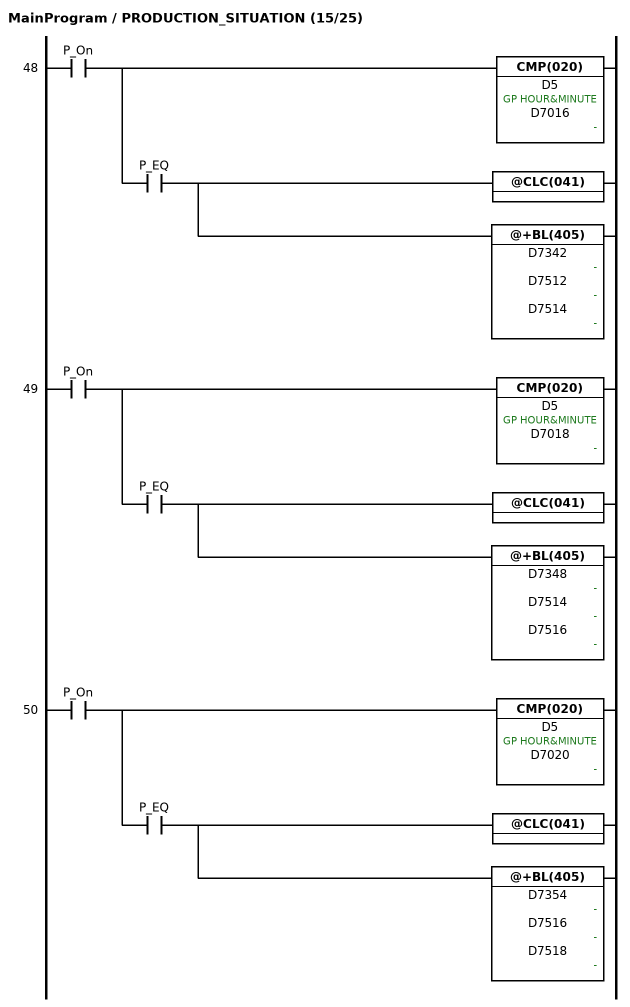
; [picture p240: MainProgram / PRODUCTION_SITUATION, rungs 48-50]
; rung 48
LD P_On
CMP(020) D5 D7016  ; GP HOUR&MINUTE, -
AND P_EQ
@CLC(041)
@+BL(405) D7342 D7512 D7514  ; -
; rung 49
LD P_On
CMP(020) D5 D7018  ; GP HOUR&MINUTE, -
AND P_EQ
@CLC(041)
@+BL(405) D7348 D7514 D7516  ; -
; rung 50
LD P_On
CMP(020) D5 D7020  ; GP HOUR&MINUTE, -
AND P_EQ
@CLC(041)
@+BL(405) D7354 D7516 D7518  ; -

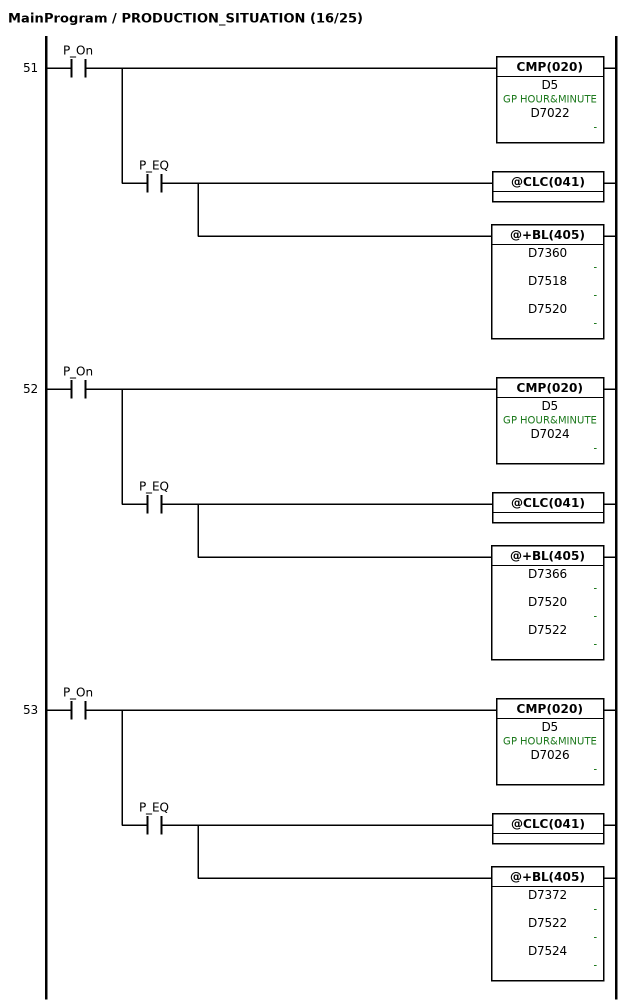
; rung 51
LD P_On
CMP(020) D5 D7022  ; GP HOUR&MINUTE, -
AND P_EQ
@CLC(041)
@+BL(405) D7360 D7518 D7520  ; -
; rung 52
LD P_On
CMP(020) D5 D7024  ; GP HOUR&MINUTE, -
AND P_EQ
@CLC(041)
@+BL(405) D7366 D7520 D7522  ; -
; rung 53
LD P_On
CMP(020) D5 D7026  ; GP HOUR&MINUTE, -
AND P_EQ
@CLC(041)
@+BL(405) D7372 D7522 D7524  ; -

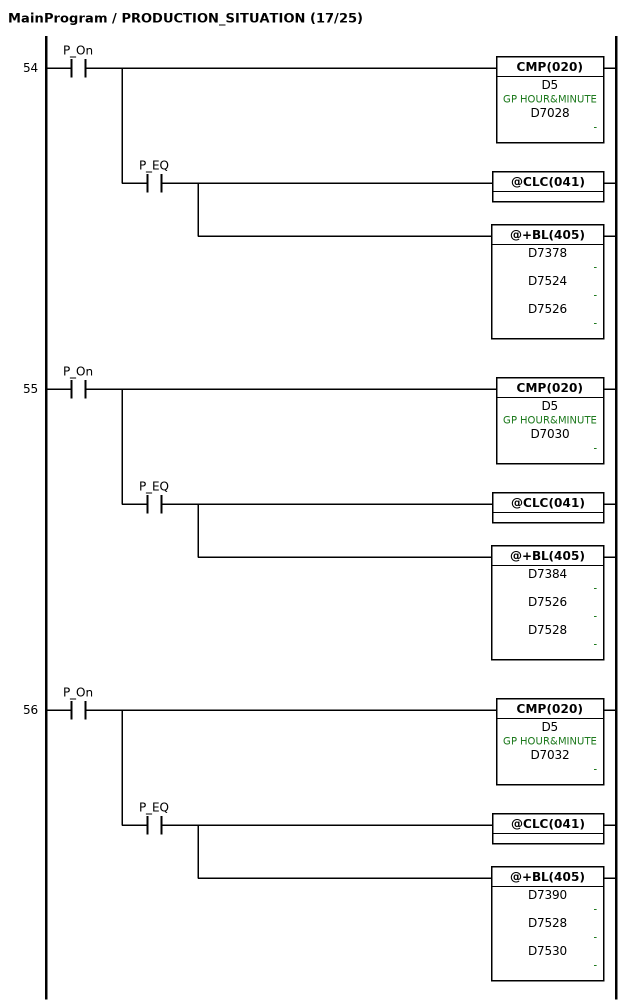
; rung 54
LD P_On
CMP(020) D5 D7028  ; GP HOUR&MINUTE, -
AND P_EQ
@CLC(041)
@+BL(405) D7378 D7524 D7526  ; -
; rung 55
LD P_On
CMP(020) D5 D7030  ; GP HOUR&MINUTE, -
AND P_EQ
@CLC(041)
@+BL(405) D7384 D7526 D7528  ; -
; rung 56
LD P_On
CMP(020) D5 D7032  ; GP HOUR&MINUTE, -
AND P_EQ
@CLC(041)
@+BL(405) D7390 D7528 D7530  ; -

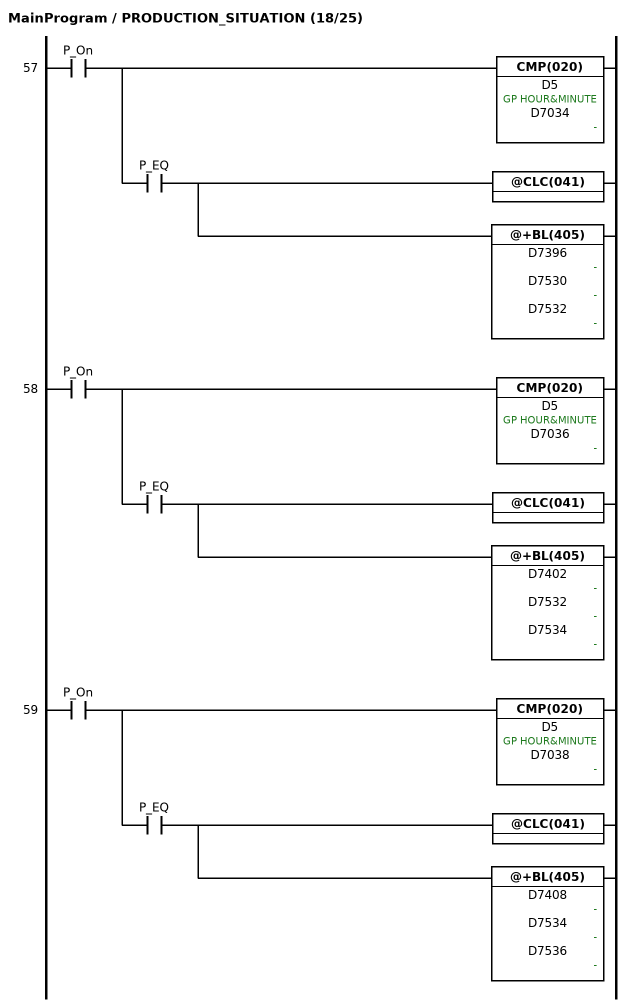
; rung 57
LD P_On
CMP(020) D5 D7034  ; GP HOUR&MINUTE, -
AND P_EQ
@CLC(041)
@+BL(405) D7396 D7530 D7532  ; -
; rung 58
LD P_On
CMP(020) D5 D7036  ; GP HOUR&MINUTE, -
AND P_EQ
@CLC(041)
@+BL(405) D7402 D7532 D7534  ; -
; rung 59
LD P_On
CMP(020) D5 D7038  ; GP HOUR&MINUTE, -
AND P_EQ
@CLC(041)
@+BL(405) D7408 D7534 D7536  ; -

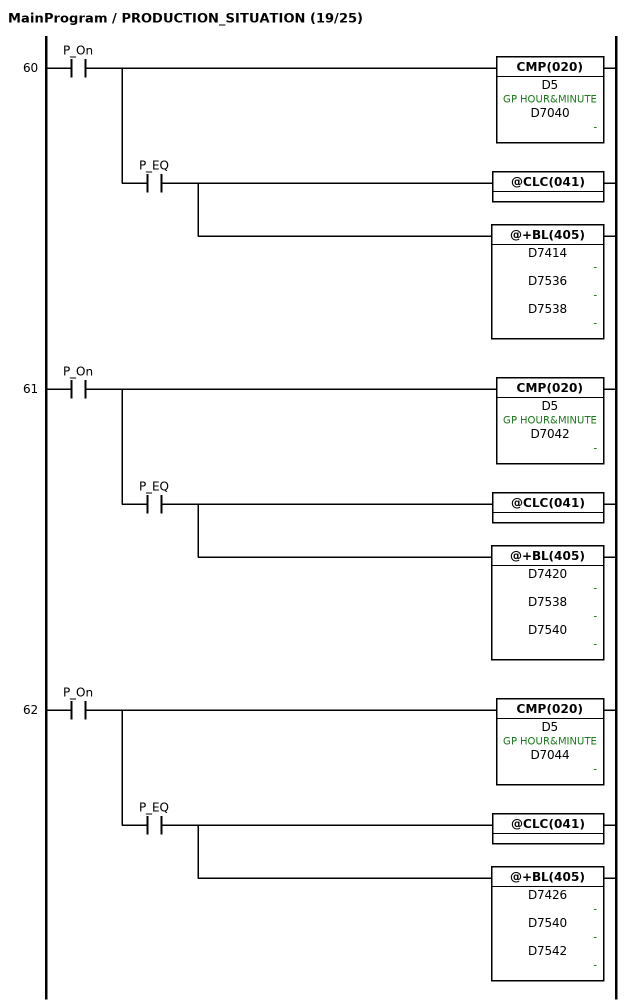
; rung 60
LD P_On
CMP(020) D5 D7040  ; GP HOUR&MINUTE, -
AND P_EQ
@CLC(041)
@+BL(405) D7414 D7536 D7538  ; -
; rung 61
LD P_On
CMP(020) D5 D7042  ; GP HOUR&MINUTE, -
AND P_EQ
@CLC(041)
@+BL(405) D7420 D7538 D7540  ; -
; rung 62
LD P_On
CMP(020) D5 D7044  ; GP HOUR&MINUTE, -
AND P_EQ
@CLC(041)
@+BL(405) D7426 D7540 D7542  ; -

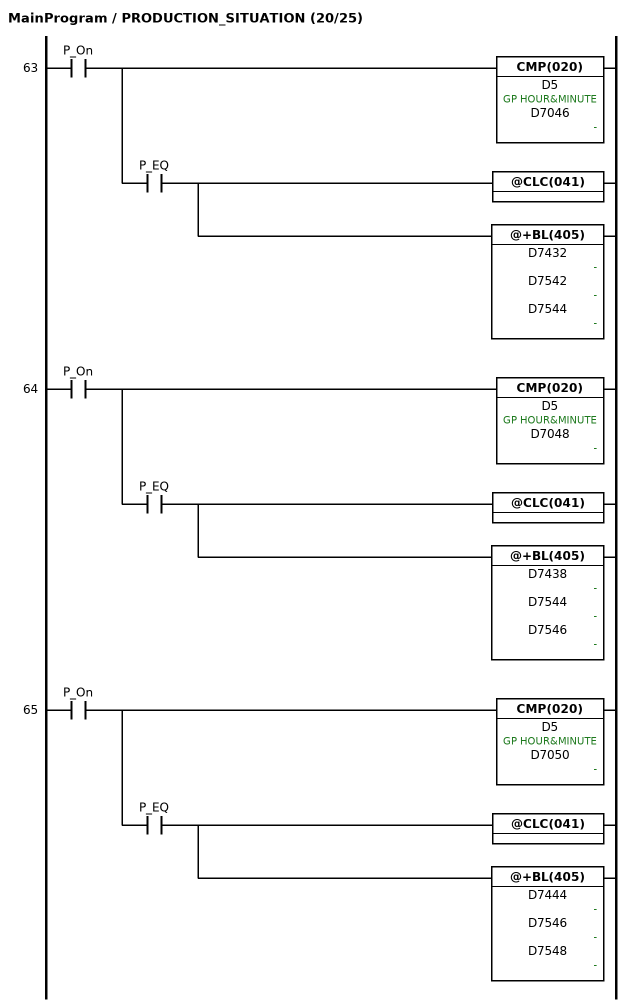
; rung 63
LD P_On
CMP(020) D5 D7046  ; GP HOUR&MINUTE, -
AND P_EQ
@CLC(041)
@+BL(405) D7432 D7542 D7544  ; -
; rung 64
LD P_On
CMP(020) D5 D7048  ; GP HOUR&MINUTE, -
AND P_EQ
@CLC(041)
@+BL(405) D7438 D7544 D7546  ; -
; rung 65
LD P_On
CMP(020) D5 D7050  ; GP HOUR&MINUTE, -
AND P_EQ
@CLC(041)
@+BL(405) D7444 D7546 D7548  ; -

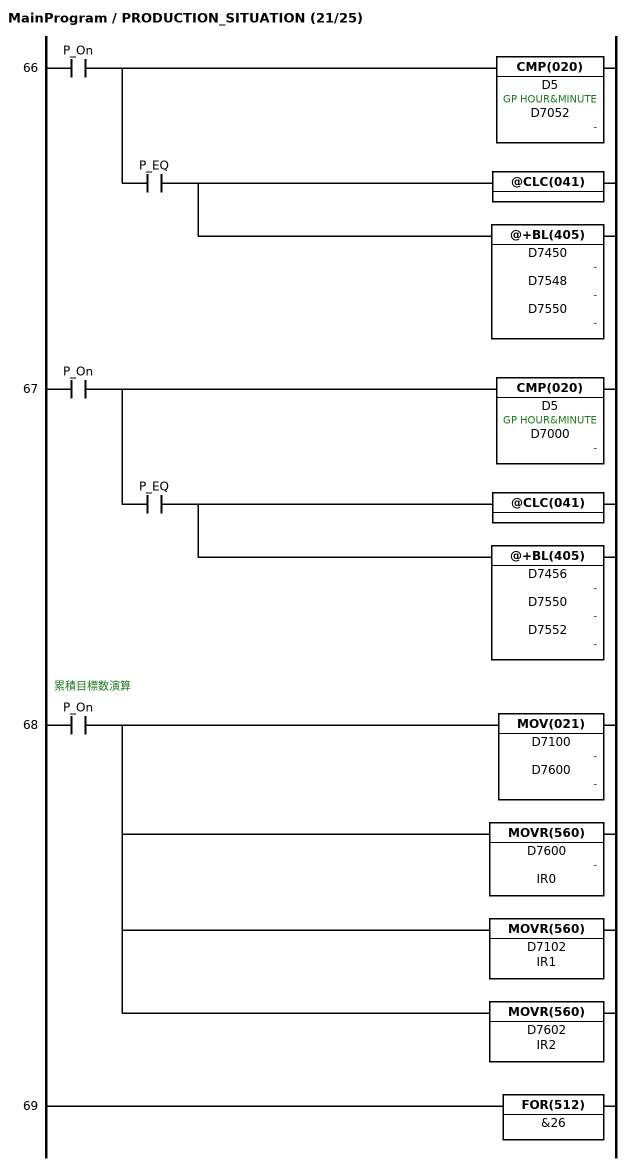
; rung 66
LD P_On
CMP(020) D5 D7052  ; GP HOUR&MINUTE, -
AND P_EQ
@CLC(041)
@+BL(405) D7450 D7548 D7550  ; -
; rung 67
LD P_On
CMP(020) D5 D7000  ; GP HOUR&MINUTE, -
AND P_EQ
@CLC(041)
@+BL(405) D7456 D7550 D7552  ; -
; rung 68: 累積目標数演算
LD P_On
MOV(021) D7100 D7600  ; -
MOVR(560) D7600 IR0  ; -
MOVR(560) D7102 IR1
MOVR(560) D7602 IR2
; rung 69
FOR(512) &26

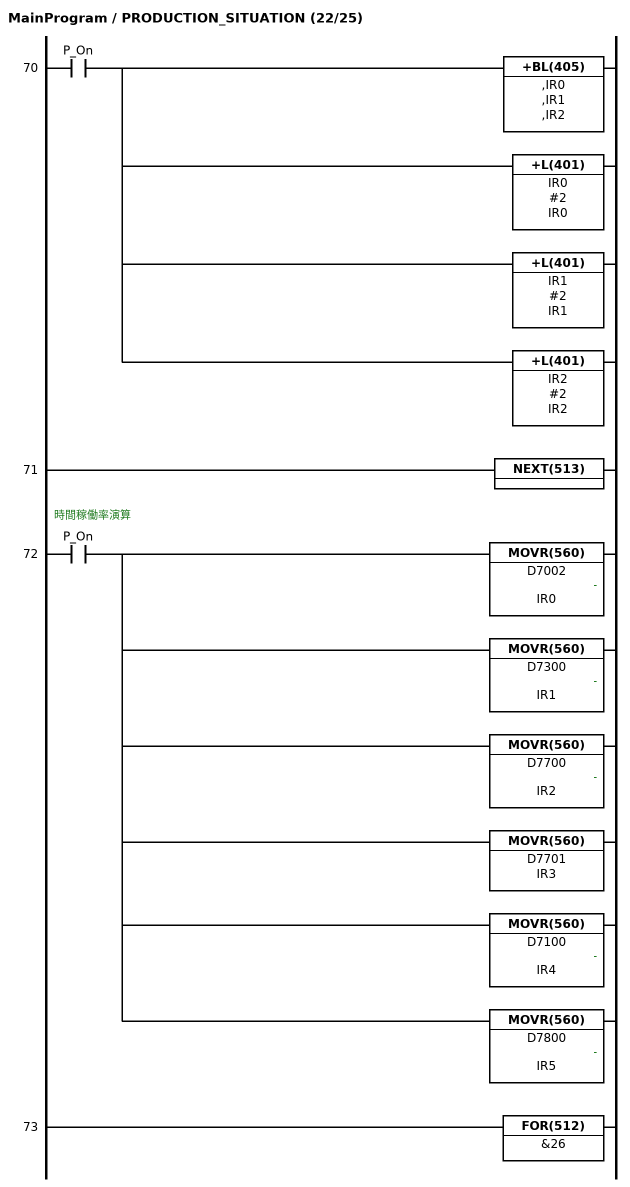
; rung 70
LD P_On
+BL(405) ,IR0 ,IR1 ,IR2
+L(401) IR0 #2 IR0
+L(401) IR1 #2 IR1
+L(401) IR2 #2 IR2
; rung 71
NEXT(513)
; rung 72: 時間稼働率演算
LD P_On
MOVR(560) D7002 IR0  ; -
MOVR(560) D7300 IR1  ; -
MOVR(560) D7700 IR2  ; -
MOVR(560) D7701 IR3
MOVR(560) D7100 IR4  ; -
MOVR(560) D7800 IR5  ; -
; rung 73
FOR(512) &26

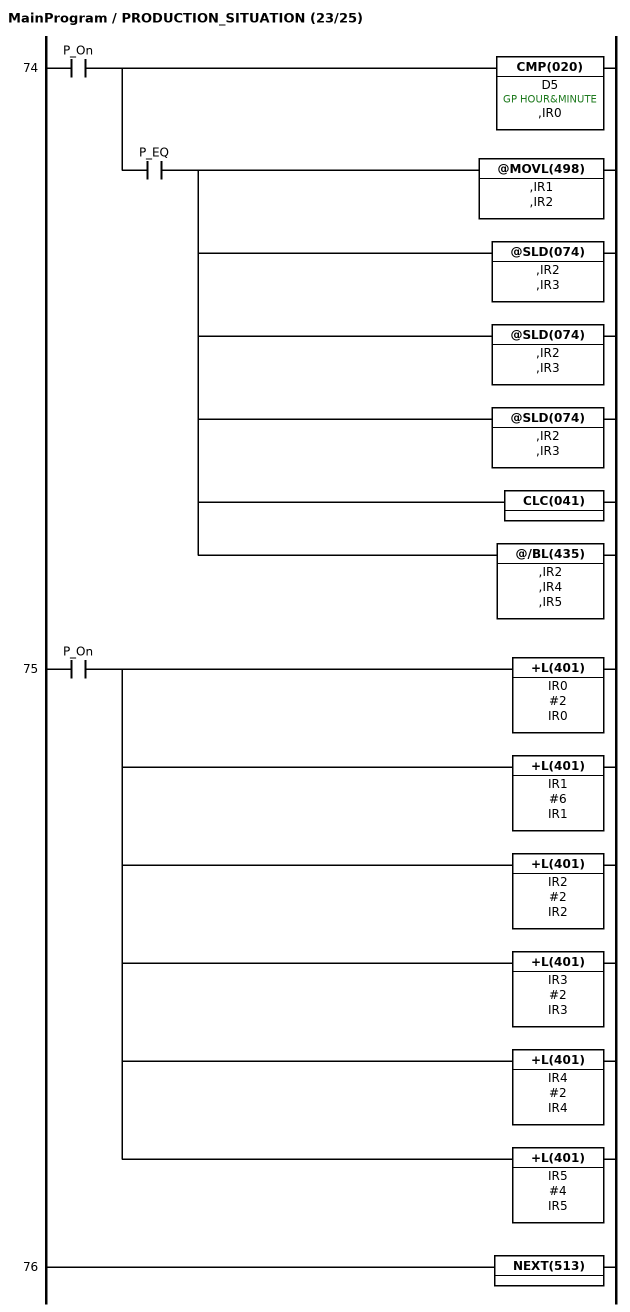
; rung 74
LD P_On
CMP(020) D5 ,IR0  ; GP HOUR&MINUTE
AND P_EQ
@MOVL(498) ,IR1 ,IR2
@SLD(074) ,IR2 ,IR3
@SLD(074) ,IR2 ,IR3
@SLD(074) ,IR2 ,IR3
CLC(041)
@/BL(435) ,IR2 ,IR4 ,IR5
; rung 75
LD P_On
+L(401) IR0 #2 IR0
+L(401) IR1 #6 IR1
+L(401) IR2 #2 IR2
+L(401) IR3 #2 IR3
+L(401) IR4 #2 IR4
+L(401) IR5 #4 IR5
; rung 76
NEXT(513)

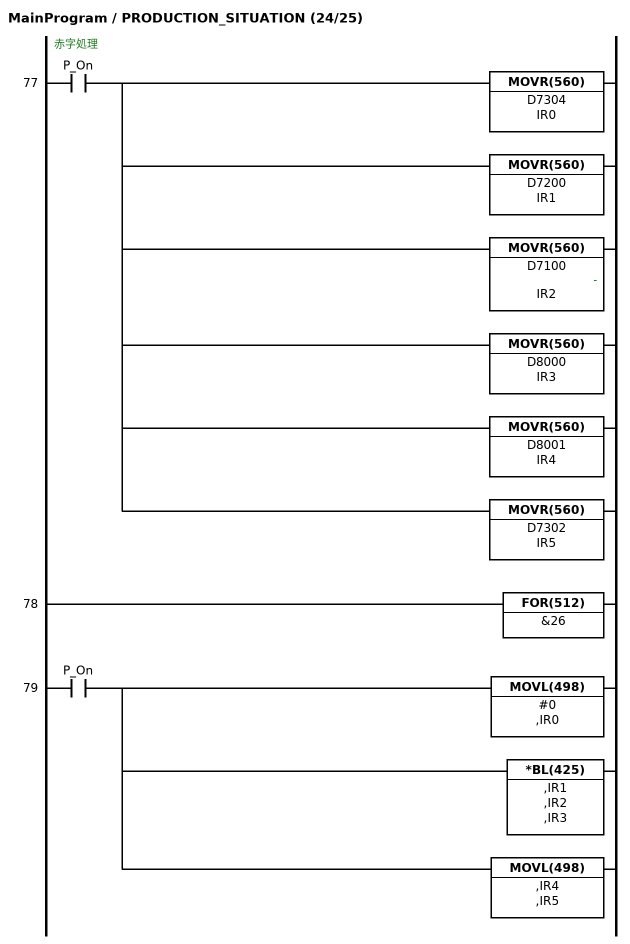
; rung 77: 赤字処理
LD P_On
MOVR(560) D7304 IR0
MOVR(560) D7200 IR1
MOVR(560) D7100 IR2  ; -
MOVR(560) D8000 IR3
MOVR(560) D8001 IR4
MOVR(560) D7302 IR5
; rung 78
FOR(512) &26
; rung 79
LD P_On
MOVL(498) #0 ,IR0
*BL(425) ,IR1 ,IR2 ,IR3
MOVL(498) ,IR4 ,IR5

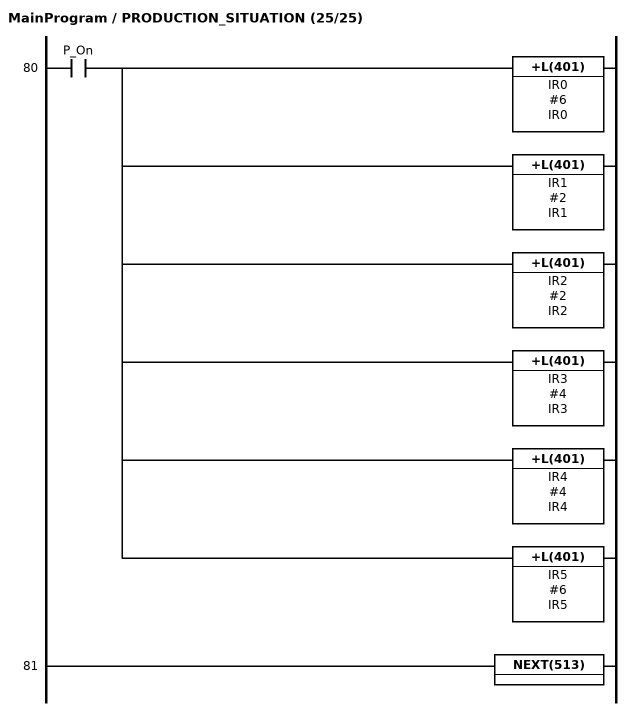
; rung 80
LD P_On
+L(401) IR0 #6 IR0
+L(401) IR1 #2 IR1
+L(401) IR2 #2 IR2
+L(401) IR3 #4 IR3
+L(401) IR4 #4 IR4
+L(401) IR5 #6 IR5
; rung 81
NEXT(513)

### Section OPERATION_RATE

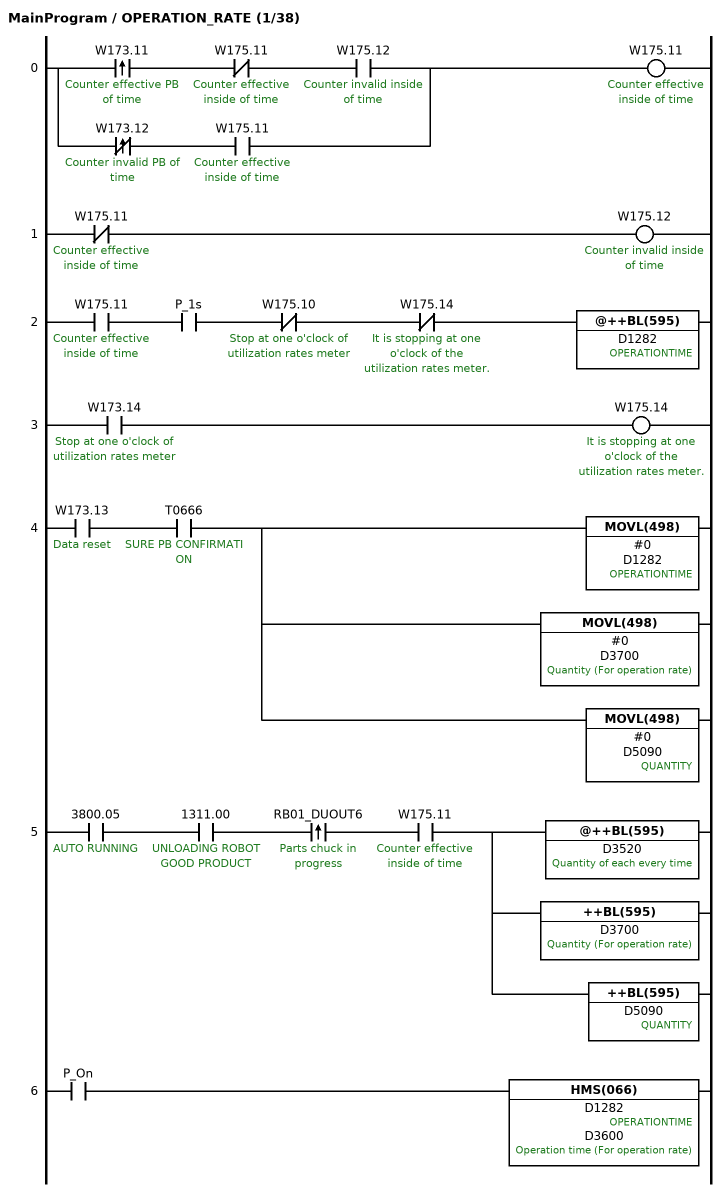
; rung 0
@LD W173.11  ; Counter effective PB of time
ANDNOT W175.11  ; Counter effective inside of time
AND W175.12  ; Counter invalid inside of time
@LDNOT W173.12  ; Counter invalid PB of time
AND W175.11  ; Counter effective inside of time
ORLD
OUT W175.11  ; Counter effective inside of time
; rung 1
LDNOT W175.11  ; Counter effective inside of time
OUT W175.12  ; Counter invalid inside of time
; rung 2
LD W175.11  ; Counter effective inside of time
AND P_1s
ANDNOT W175.10  ; Stop at one o'clock of utilization rates meter
ANDNOT W175.14  ; It is stopping at one o'clock of the utilization rates meter.
@++BL(595) D1282  ; OPERATIONTIME
; rung 3
LD W173.14  ; Stop at one o'clock of utilization rates meter
OUT W175.14  ; It is stopping at one o'clock of the utilization rates meter.
; rung 4
LD W173.13  ; Data reset
AND T0666  ; SURE PB CONFIRMATION
MOVL(498) #0 D1282  ; OPERATIONTIME
MOVL(498) #0 D3700  ; Quantity (For operation rate)
MOVL(498) #0 D5090  ; QUANTITY
; rung 5
LD 3800.05  ; AUTO RUNNING
AND 1311.00  ; UNLOADING ROBOT GOOD PRODUCT
@AND RB01_DUOUT6  ; Parts chuck in progress
AND W175.11  ; Counter effective inside of time
@++BL(595) D3520  ; Quantity of each every time
++BL(595) D3700  ; Quantity (For operation rate)
++BL(595) D5090  ; QUANTITY
; rung 6
LD P_On
HMS(066) D1282 D3600  ; OPERATIONTIME, Operation time (For operation rate)

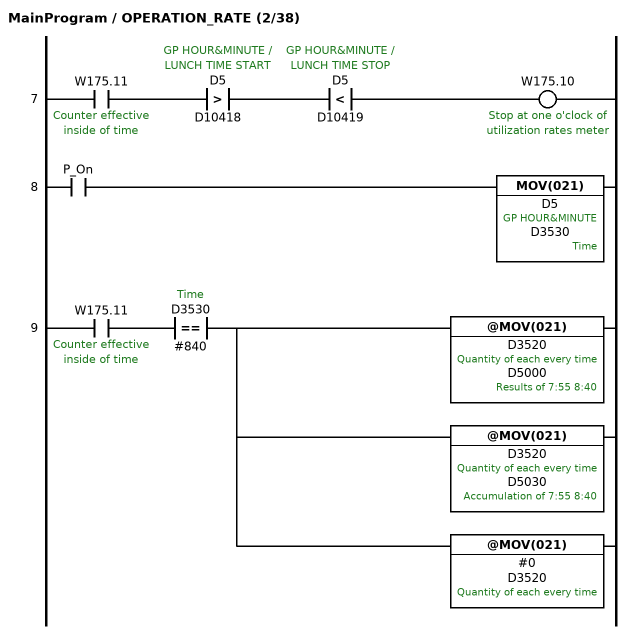
; rung 7
LD W175.11  ; Counter effective inside of time
AND>(320) D5 D10418  ; GP HOUR&MINUTE, LUNCH TIME START
AND<(310) D5 D10419  ; GP HOUR&MINUTE, LUNCH TIME STOP
OUT W175.10  ; Stop at one o'clock of utilization rates meter
; rung 8
LD P_On
MOV(021) D5 D3530  ; GP HOUR&MINUTE, Time
; rung 9
LD W175.11  ; Counter effective inside of time
AND=L(301) D3530 #840  ; Time
@MOV(021) D3520 D5000  ; Quantity of each every time, Results of 7:55 8:40
@MOV(021) D3520 D5030  ; Quantity of each every time, Accumulation of 7:55 8:40
@MOV(021) #0 D3520  ; Quantity of each every time

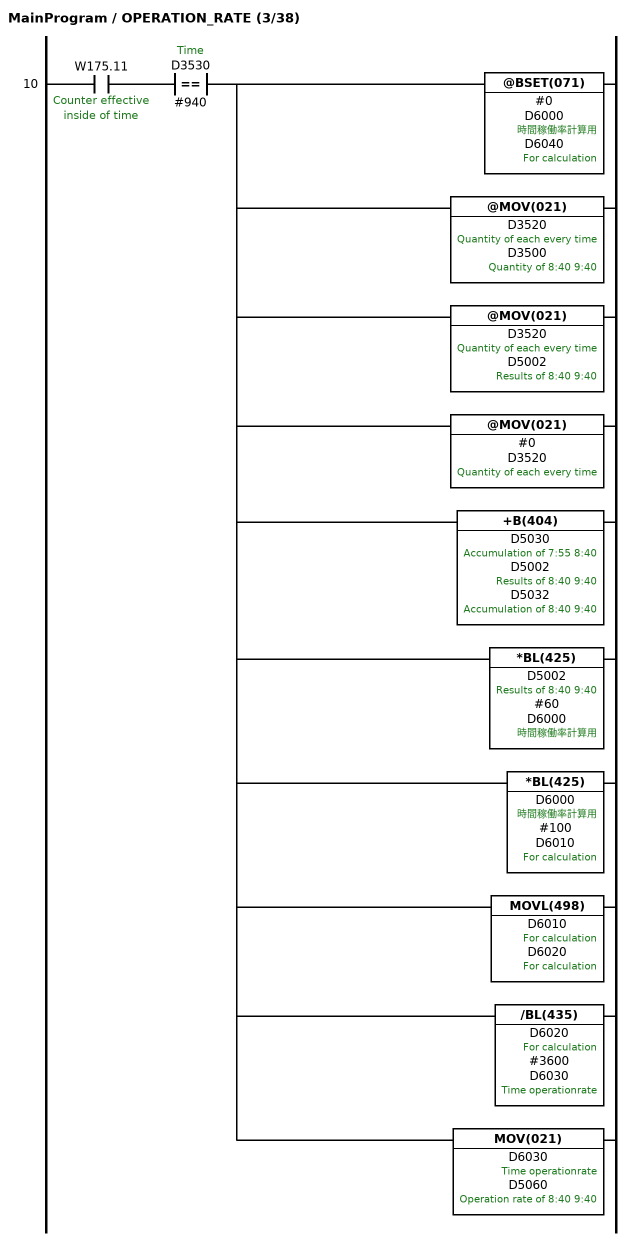
; rung 10
LD W175.11  ; Counter effective inside of time
AND=L(301) D3530 #940  ; Time
@BSET(071) #0 D6000 D6040  ; 時間稼働率計算用, For calculation
@MOV(021) D3520 D3500  ; Quantity of each every time, Quantity of 8:40 9:40
@MOV(021) D3520 D5002  ; Quantity of each every time, Results of 8:40 9:40
@MOV(021) #0 D3520  ; Quantity of each every time
+B(404) D5030 D5002 D5032  ; Accumulation of 7:55 8:40, Results of 8:40 9:40, Accumulation of 8:40 9:40
*BL(425) D5002 #60 D6000  ; Results of 8:40 9:40, 時間稼働率計算用
*BL(425) D6000 #100 D6010  ; 時間稼働率計算用, For calculation
MOVL(498) D6010 D6020  ; For calculation
/BL(435) D6020 #3600 D6030  ; For calculation, Time operationrate
MOV(021) D6030 D5060  ; Time operationrate, Operation rate of 8:40 9:40

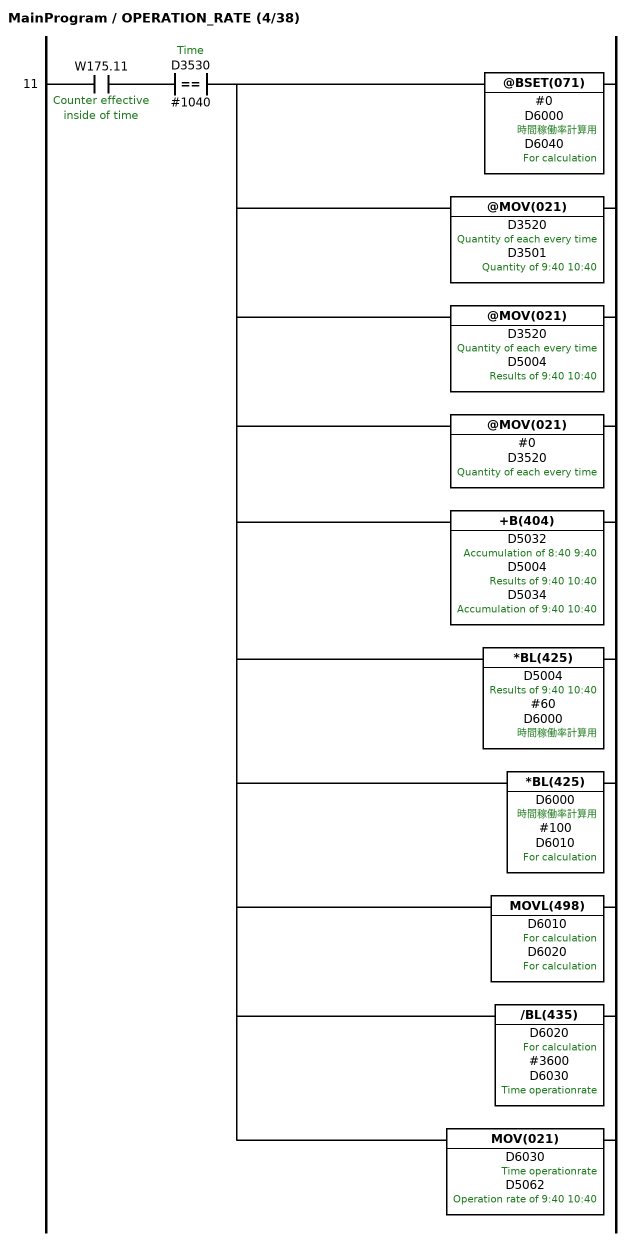
; rung 11
LD W175.11  ; Counter effective inside of time
AND=L(301) D3530 #1040  ; Time
@BSET(071) #0 D6000 D6040  ; 時間稼働率計算用, For calculation
@MOV(021) D3520 D3501  ; Quantity of each every time, Quantity of 9:40 10:40
@MOV(021) D3520 D5004  ; Quantity of each every time, Results of 9:40 10:40
@MOV(021) #0 D3520  ; Quantity of each every time
+B(404) D5032 D5004 D5034  ; Accumulation of 8:40 9:40, Results of 9:40 10:40, Accumulation of 9:40 10:40
*BL(425) D5004 #60 D6000  ; Results of 9:40 10:40, 時間稼働率計算用
*BL(425) D6000 #100 D6010  ; 時間稼働率計算用, For calculation
MOVL(498) D6010 D6020  ; For calculation
/BL(435) D6020 #3600 D6030  ; For calculation, Time operationrate
MOV(021) D6030 D5062  ; Time operationrate, Operation rate of 9:40 10:40

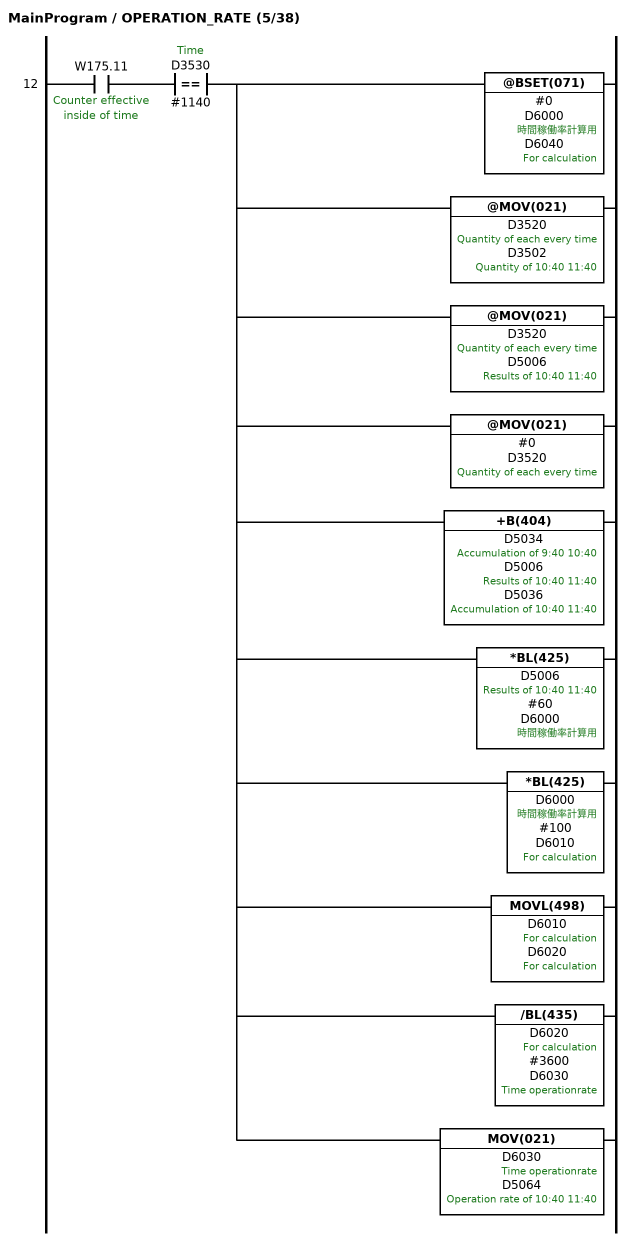
; rung 12
LD W175.11  ; Counter effective inside of time
AND=L(301) D3530 #1140  ; Time
@BSET(071) #0 D6000 D6040  ; 時間稼働率計算用, For calculation
@MOV(021) D3520 D3502  ; Quantity of each every time, Quantity of 10:40 11:40
@MOV(021) D3520 D5006  ; Quantity of each every time, Results of 10:40 11:40
@MOV(021) #0 D3520  ; Quantity of each every time
+B(404) D5034 D5006 D5036  ; Accumulation of 9:40 10:40, Results of 10:40 11:40, Accumulation of 10:40 11:40
*BL(425) D5006 #60 D6000  ; Results of 10:40 11:40, 時間稼働率計算用
*BL(425) D6000 #100 D6010  ; 時間稼働率計算用, For calculation
MOVL(498) D6010 D6020  ; For calculation
/BL(435) D6020 #3600 D6030  ; For calculation, Time operationrate
MOV(021) D6030 D5064  ; Time operationrate, Operation rate of 10:40 11:40

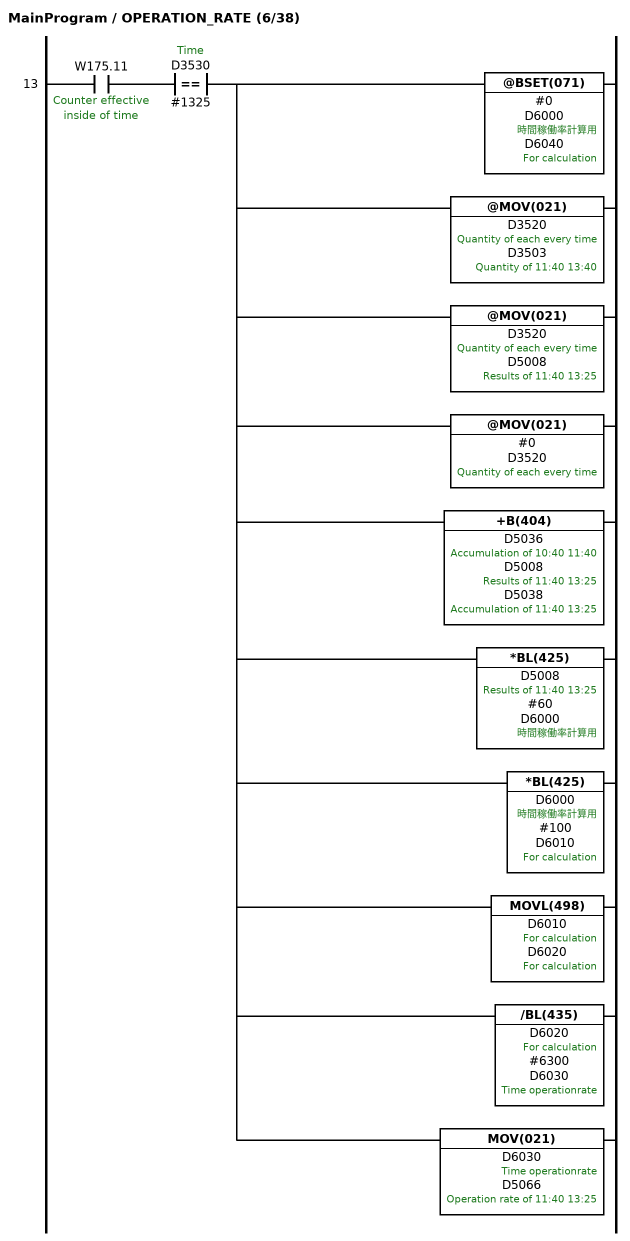
; rung 13
LD W175.11  ; Counter effective inside of time
AND=L(301) D3530 #1325  ; Time
@BSET(071) #0 D6000 D6040  ; 時間稼働率計算用, For calculation
@MOV(021) D3520 D3503  ; Quantity of each every time, Quantity of 11:40 13:40
@MOV(021) D3520 D5008  ; Quantity of each every time, Results of 11:40 13:25
@MOV(021) #0 D3520  ; Quantity of each every time
+B(404) D5036 D5008 D5038  ; Accumulation of 10:40 11:40, Results of 11:40 13:25, Accumulation of 11:40 13:25
*BL(425) D5008 #60 D6000  ; Results of 11:40 13:25, 時間稼働率計算用
*BL(425) D6000 #100 D6010  ; 時間稼働率計算用, For calculation
MOVL(498) D6010 D6020  ; For calculation
/BL(435) D6020 #6300 D6030  ; For calculation, Time operationrate
MOV(021) D6030 D5066  ; Time operationrate, Operation rate of 11:40 13:25

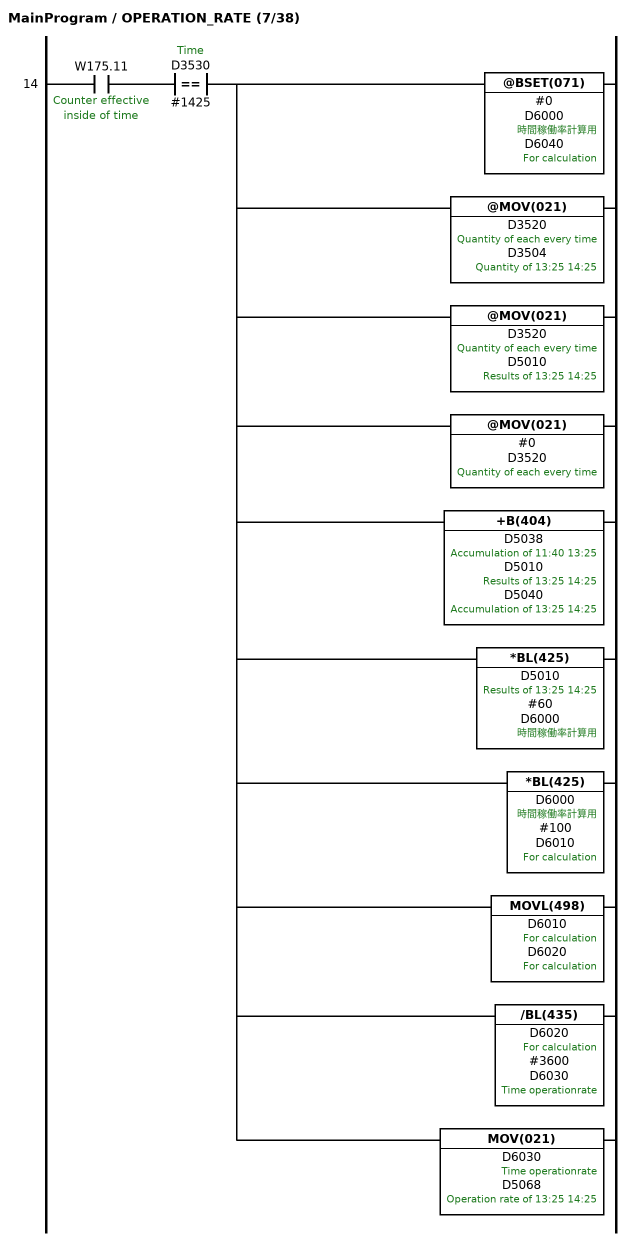
; rung 14
LD W175.11  ; Counter effective inside of time
AND=L(301) D3530 #1425  ; Time
@BSET(071) #0 D6000 D6040  ; 時間稼働率計算用, For calculation
@MOV(021) D3520 D3504  ; Quantity of each every time, Quantity of 13:25 14:25
@MOV(021) D3520 D5010  ; Quantity of each every time, Results of 13:25 14:25
@MOV(021) #0 D3520  ; Quantity of each every time
+B(404) D5038 D5010 D5040  ; Accumulation of 11:40 13:25, Results of 13:25 14:25, Accumulation of 13:25 14:25
*BL(425) D5010 #60 D6000  ; Results of 13:25 14:25, 時間稼働率計算用
*BL(425) D6000 #100 D6010  ; 時間稼働率計算用, For calculation
MOVL(498) D6010 D6020  ; For calculation
/BL(435) D6020 #3600 D6030  ; For calculation, Time operationrate
MOV(021) D6030 D5068  ; Time operationrate, Operation rate of 13:25 14:25

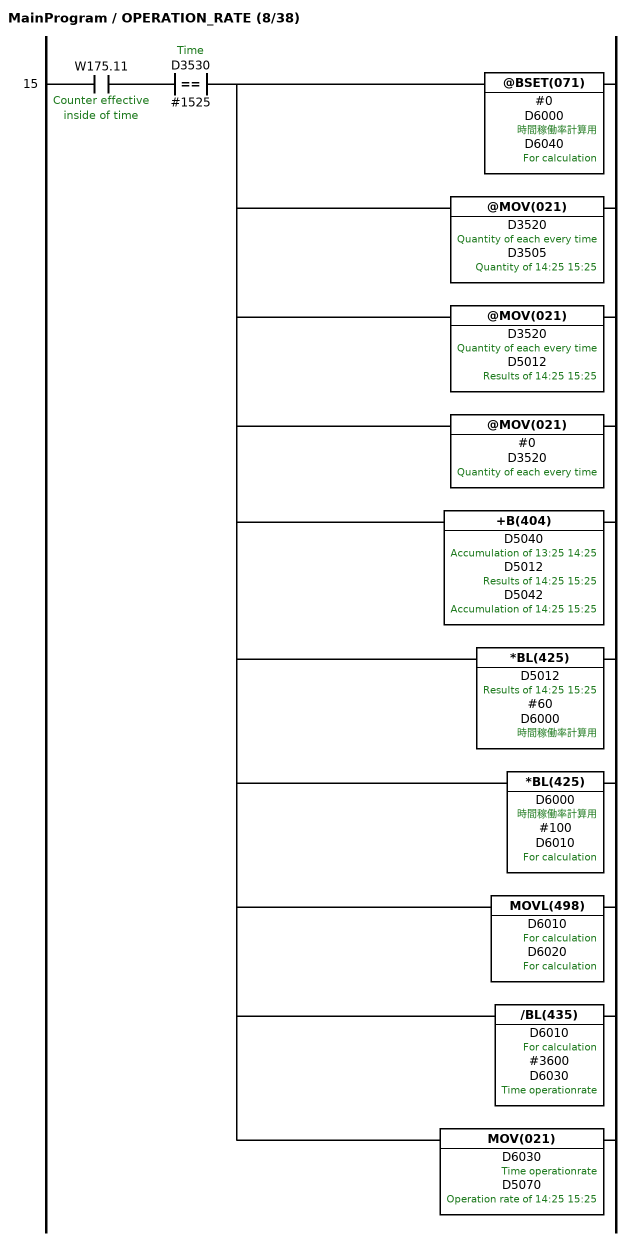
; rung 15
LD W175.11  ; Counter effective inside of time
AND=L(301) D3530 #1525  ; Time
@BSET(071) #0 D6000 D6040  ; 時間稼働率計算用, For calculation
@MOV(021) D3520 D3505  ; Quantity of each every time, Quantity of 14:25 15:25
@MOV(021) D3520 D5012  ; Quantity of each every time, Results of 14:25 15:25
@MOV(021) #0 D3520  ; Quantity of each every time
+B(404) D5040 D5012 D5042  ; Accumulation of 13:25 14:25, Results of 14:25 15:25, Accumulation of 14:25 15:25
*BL(425) D5012 #60 D6000  ; Results of 14:25 15:25, 時間稼働率計算用
*BL(425) D6000 #100 D6010  ; 時間稼働率計算用, For calculation
MOVL(498) D6010 D6020  ; For calculation
/BL(435) D6010 #3600 D6030  ; For calculation, Time operationrate
MOV(021) D6030 D5070  ; Time operationrate, Operation rate of 14:25 15:25

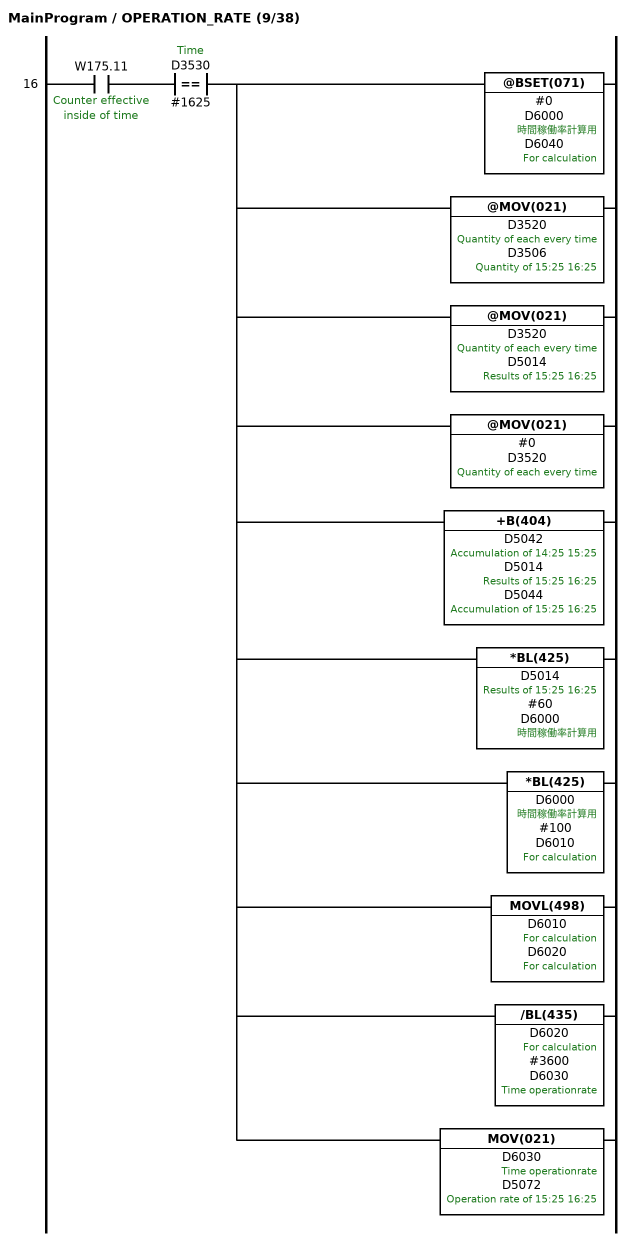
; rung 16
LD W175.11  ; Counter effective inside of time
AND=L(301) D3530 #1625  ; Time
@BSET(071) #0 D6000 D6040  ; 時間稼働率計算用, For calculation
@MOV(021) D3520 D3506  ; Quantity of each every time, Quantity of 15:25 16:25
@MOV(021) D3520 D5014  ; Quantity of each every time, Results of 15:25 16:25
@MOV(021) #0 D3520  ; Quantity of each every time
+B(404) D5042 D5014 D5044  ; Accumulation of 14:25 15:25, Results of 15:25 16:25, Accumulation of 15:25 16:25
*BL(425) D5014 #60 D6000  ; Results of 15:25 16:25, 時間稼働率計算用
*BL(425) D6000 #100 D6010  ; 時間稼働率計算用, For calculation
MOVL(498) D6010 D6020  ; For calculation
/BL(435) D6020 #3600 D6030  ; For calculation, Time operationrate
MOV(021) D6030 D5072  ; Time operationrate, Operation rate of 15:25 16:25

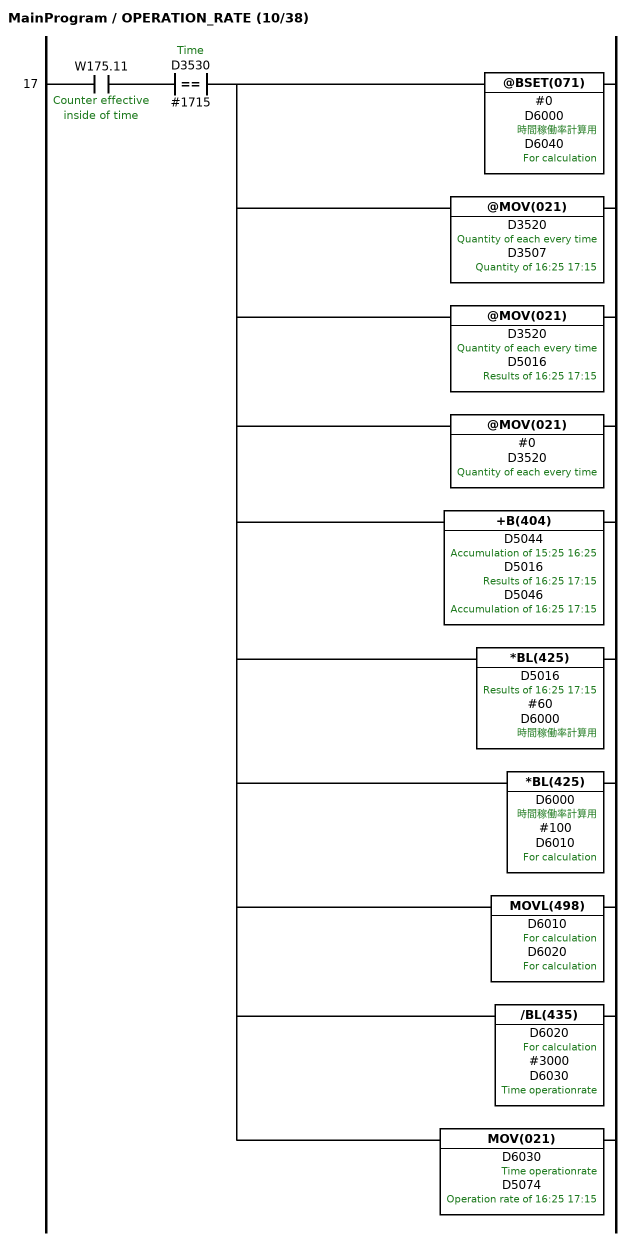
; rung 17
LD W175.11  ; Counter effective inside of time
AND=L(301) D3530 #1715  ; Time
@BSET(071) #0 D6000 D6040  ; 時間稼働率計算用, For calculation
@MOV(021) D3520 D3507  ; Quantity of each every time, Quantity of 16:25 17:15
@MOV(021) D3520 D5016  ; Quantity of each every time, Results of 16:25 17:15
@MOV(021) #0 D3520  ; Quantity of each every time
+B(404) D5044 D5016 D5046  ; Accumulation of 15:25 16:25, Results of 16:25 17:15, Accumulation of 16:25 17:15
*BL(425) D5016 #60 D6000  ; Results of 16:25 17:15, 時間稼働率計算用
*BL(425) D6000 #100 D6010  ; 時間稼働率計算用, For calculation
MOVL(498) D6010 D6020  ; For calculation
/BL(435) D6020 #3000 D6030  ; For calculation, Time operationrate
MOV(021) D6030 D5074  ; Time operationrate, Operation rate of 16:25 17:15

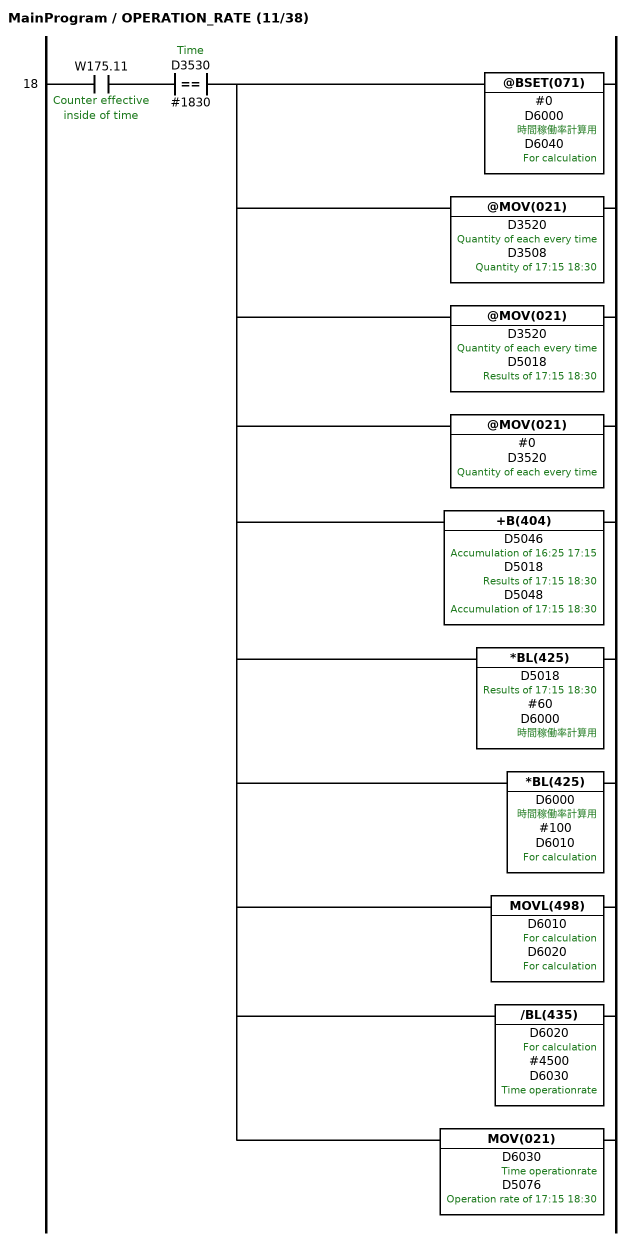
; rung 18
LD W175.11  ; Counter effective inside of time
AND=L(301) D3530 #1830  ; Time
@BSET(071) #0 D6000 D6040  ; 時間稼働率計算用, For calculation
@MOV(021) D3520 D3508  ; Quantity of each every time, Quantity of 17:15 18:30
@MOV(021) D3520 D5018  ; Quantity of each every time, Results of 17:15 18:30
@MOV(021) #0 D3520  ; Quantity of each every time
+B(404) D5046 D5018 D5048  ; Accumulation of 16:25 17:15, Results of 17:15 18:30, Accumulation of 17:15 18:30
*BL(425) D5018 #60 D6000  ; Results of 17:15 18:30, 時間稼働率計算用
*BL(425) D6000 #100 D6010  ; 時間稼働率計算用, For calculation
MOVL(498) D6010 D6020  ; For calculation
/BL(435) D6020 #4500 D6030  ; For calculation, Time operationrate
MOV(021) D6030 D5076  ; Time operationrate, Operation rate of 17:15 18:30

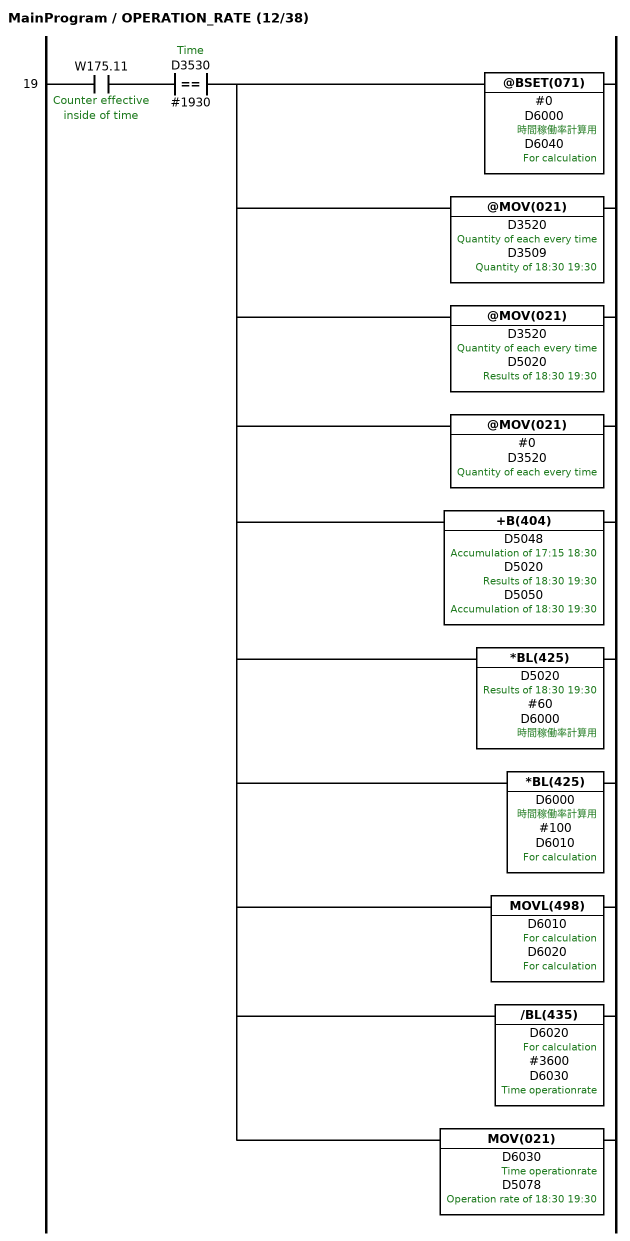
; rung 19
LD W175.11  ; Counter effective inside of time
AND=L(301) D3530 #1930  ; Time
@BSET(071) #0 D6000 D6040  ; 時間稼働率計算用, For calculation
@MOV(021) D3520 D3509  ; Quantity of each every time, Quantity of 18:30 19:30
@MOV(021) D3520 D5020  ; Quantity of each every time, Results of 18:30 19:30
@MOV(021) #0 D3520  ; Quantity of each every time
+B(404) D5048 D5020 D5050  ; Accumulation of 17:15 18:30, Results of 18:30 19:30, Accumulation of 18:30 19:30
*BL(425) D5020 #60 D6000  ; Results of 18:30 19:30, 時間稼働率計算用
*BL(425) D6000 #100 D6010  ; 時間稼働率計算用, For calculation
MOVL(498) D6010 D6020  ; For calculation
/BL(435) D6020 #3600 D6030  ; For calculation, Time operationrate
MOV(021) D6030 D5078  ; Time operationrate, Operation rate of 18:30 19:30

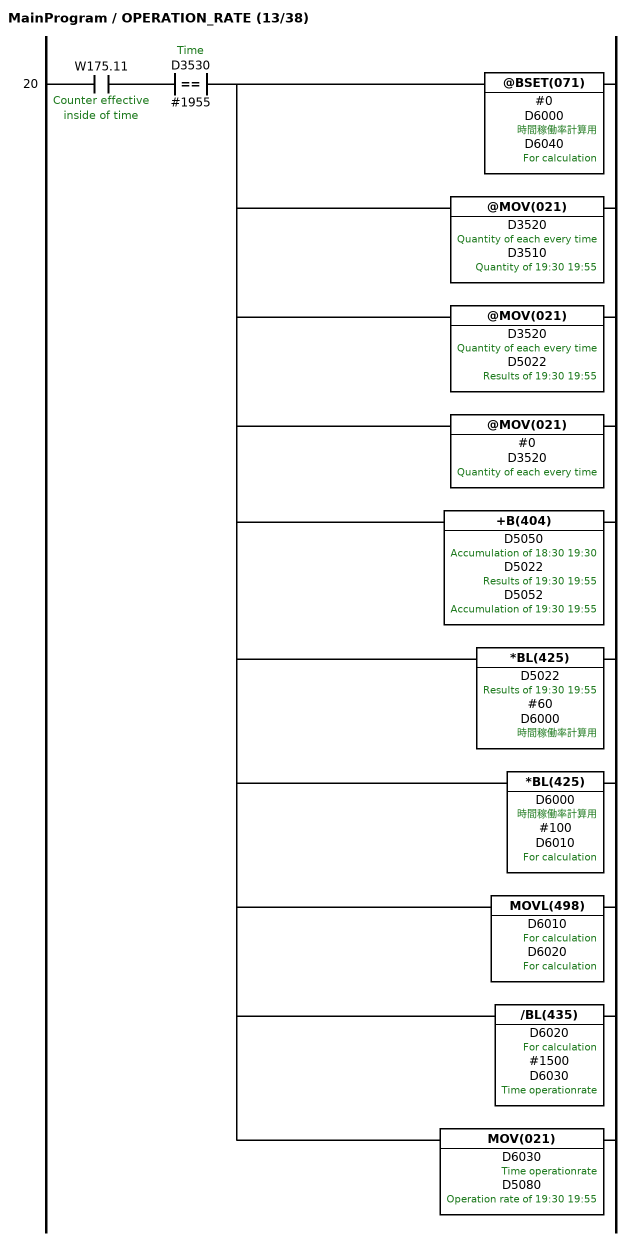
; rung 20
LD W175.11  ; Counter effective inside of time
AND=L(301) D3530 #1955  ; Time
@BSET(071) #0 D6000 D6040  ; 時間稼働率計算用, For calculation
@MOV(021) D3520 D3510  ; Quantity of each every time, Quantity of 19:30 19:55
@MOV(021) D3520 D5022  ; Quantity of each every time, Results of 19:30 19:55
@MOV(021) #0 D3520  ; Quantity of each every time
+B(404) D5050 D5022 D5052  ; Accumulation of 18:30 19:30, Results of 19:30 19:55, Accumulation of 19:30 19:55
*BL(425) D5022 #60 D6000  ; Results of 19:30 19:55, 時間稼働率計算用
*BL(425) D6000 #100 D6010  ; 時間稼働率計算用, For calculation
MOVL(498) D6010 D6020  ; For calculation
/BL(435) D6020 #1500 D6030  ; For calculation, Time operationrate
MOV(021) D6030 D5080  ; Time operationrate, Operation rate of 19:30 19:55

